TYPE ST_ControlElement_HMI_Link_1 EXTENDS ST_BaseControlElement_HMI_Link :
STRUCT
	stControlElement			: ST_ControlElement_HMI_1;
	
	stComponent1				: ST_Component_HMI_Link;
	stComponent2				: ST_Component_HMI_Link;
	
END_STRUCT
END_TYPE

(* stored: Version 1.1.0.1, ProductVersion 3.1.4024.15
   DUT ST_ControlElement_HMI_Link_1: Id {a2ca18d4-d91f-4e2a-9bb8-df92e9dfc9ce} *)
